(* Coast stop, Quick stop, Ramp stop *)
	IF fbProfidriveGSM.eState = E_ProfidriveGSM_State.S1_SwitchingOnInhibited THEN
		fbMoveVelocity.fTargetVelocity	:= 0;
		fbMoveVelocity.fAccMax 			:= fDecelerationCoastStop;
		fbMoveVelocity.fDecMax 			:= fDecelerationCoastStop;
	ELSIF fbProfidriveGSM.eState = E_ProfidriveGSM_State.S52_QuickStop THEN
		fbMoveVelocity.fTargetVelocity	:= 0;
		fbMoveVelocity.fAccMax 			:= fDecelerationQuickStop;
		fbMoveVelocity.fDecMax 			:= fDecelerationQuickStop;
	ELSIF fbProfidriveGSM.eState = E_ProfidriveGSM_State.S51_RampStop THEN
		fbMoveVelocity.fTargetVelocity	:= 0;
		fbMoveVelocity.fAccMax 			:= fDeceleration;
		fbMoveVelocity.fDecMax 			:= fDeceleration;
	END_IF

(* Call MoveVelocity *)
	fbMoveVelocity();
	
(* Status word *)
	stStatus.bReadyForSwitchingOn			:= fbProfidriveGSM.stStatus.b0_ReadyToSwitchOn;	
	stStatus.bReadyForOperation				:= fbProfidriveGSM.stStatus.b1_ReadyForOperation;
	stStatus.bOperationEnabled				:= stControl.bEnableOperation;
	stStatus.bFaultPresent					:= bFaultPresent;
	stStatus.bNoCoastDownActive				:= fbProfidriveGSM.eState <> E_ProfidriveGSM_State.S1_SwitchingOnInhibited;
	stStatus.bNoQuickStopActive				:= fbProfidriveGSM.eState <> E_ProfidriveGSM_State.S52_QuickStop;
	stStatus.bSwitchingOnInhibited			:= fbProfidriveGSM.stStatus.b6_SwitchingOnInhibited;
	stStatus.bAlarmPresent					:= bAlarmPresent;
	stStatus.bDeviationWithinTolerance		:= TRUE;
	stStatus.bControlRequested				:= stConfig.bControlRequested;	
	stStatus.bFrequencyLimitOk				:= TRUE;	
	stStatus.bBusy							:= ABS(fbMoveVelocity.fVelocity) > 0;
	stStatus.bInverterError					:= bInverterError;	
	stStatus.bVoltageError					:= bVoltageError;
	stStatus.bMomentError					:= bMomentError;
	stStatus.bTimerError					:= bTimerError;

(* Reset quickstop from extern *)
	IF stControl.bAcknowledgeFaults THEN
		bQuickStopExternal := FALSE;
	END_IF

(* Calculate NIST *)
	IF stConfig.fP2000 = 0 THEN
		stStatus.nIst	:= 0;
	ELSE
		stStatus.nIst	:=	REAL_TO_INT((ABS(fbMoveVelocity.fVelocity) * 16#4000) / stConfig.fP2000);
	END_IF

(* Output of actual value *)	
	IF stConfig.bOutputVelocity THEN
		ControlData := fbMoveVelocity.fVelocity;
	ELSE
		ControlData := ControlData + fbMoveVelocity.fVelocity *  GVL_Core.fbSystem.fDeltaTime * GVL_Core.fbSystem.fTimeScaling;
	END_IF
	
	fValue := ControlData;
END_METHOD

METHOD INTERNAL EvaluateParameters
VAR_INPUT
END_VAR
IF stConfig.fP1120 > 0 THEN
	fAcceleration := stConfig.fP2000/stConfig.fP1120;
ELSE
	fAcceleration := 1000;
END_IF

IF stConfig.fP1121 > 0 THEN
	fDeceleration := stConfig.fP2000/stConfig.fP1121;
ELSE
	fDeceleration := 1000;
END_IF

IF stConfig.fP1135 > 0 THEN
	fDecelerationQuickStop := stConfig.fP2000/stConfig.fP1135;
ELSE
	fDecelerationQuickStop := 1000;
END_IF

IF stConfig.fRampDownTimeCoastStop > 0 THEN
	fDecelerationCoastStop := stConfig.fP2000/stConfig.fRampDownTimeCoastStop;
ELSE
	fDecelerationCoastStop := 1000;
END_IF
END_METHOD

METHOD PUBLIC GetAcylicParameter : BOOL
VAR_INPUT
	stParameter : POINTER TO ST_PROFIdriveParam;
END_VAR
IF stParameter^.nNumber = 35 THEN
	stParameter^.nFormat := E_PROFIdriveParamFormat.FLOAT;
	stParameter^.nElements := 1;
	memcpy(ADR(stParameter^.aValue), ADR(stConfig.nR0035), 4);
END_IF
END_METHOD

METHOD INTERNAL InitRun : BOOL
VAR_INST
	bInitRun : BOOL := TRUE;
END_VAR
IF NOT bInitRun THEN RETURN; END_IF
bInitRun := FALSE;

IF pFromBus = 0 OR pToBus = 0 THEN
	ADSLOGSTR(ADSLOG_MSGTYPE_WARN, CONCAT(sPath, ': %s'), 'Plc address not set.');
END_IF
END_METHOD

METHOD INTERNAL ReadBus
VAR_INPUT
END_VAR
IF pFromBus = 0 THEN
	RETURN;
END_IF

IF NOT stConfig.bSwapProcessData THEN
	(* Control word *)
		stControl.bOFF1							:= pFromBus[0].0;
		stControl.bOFF2							:= pFromBus[0].1;
		stControl.bOFF3							:= pFromBus[0].2;
		stControl.bEnableOperation			    	:= pFromBus[0].3;
		stControl.bOperatingCondition				:= pFromBus[0].4;
		stControl.bContinueRampFunctionGenerator	:= pFromBus[0].5;
		stControl.bEnableSetpoint  				:= pFromBus[0].6;
		stControl.bAcknowledgeFaults				:= pFromBus[0].7;
		stControl.bJog1							:= pFromBus[1].0;
		stControl.bJog2							:= pFromBus[1].1;
		stControl.bDataValid						:= pFromBus[1].2;
		stControl.bFreqCorrDown					:= pFromBus[1].3;
		stControl.bFreqCorrUp						:= pFromBus[1].4;
		stControl.bParameterSelectionLSB			:= pFromBus[1].5;
		stControl.bParameterSelectionMSB			:= pFromBus[1].6;
		stControl.bReversing						:= pFromBus[1].7;
		
	(* Setpoint speed *)
		stControl.nSoll							:= UINT_TO_INT(pFromBus[2] + pFromBus[3] * 16#100);
ELSE
	(* Control word *)
		stControl.bOFF1							:= pFromBus[1].0;
		stControl.bOFF2							:= pFromBus[1].1;
		stControl.bOFF3							:= pFromBus[1].2;
		stControl.bEnableOperation				    := pFromBus[1].3;
		stControl.bOperatingCondition				:= pFromBus[1].4;
		stControl.bContinueRampFunctionGenerator	:= pFromBus[1].5;
		stControl.bEnableSetpoint  				:= pFromBus[1].6;
		stControl.bAcknowledgeFaults				:= pFromBus[1].7;
		stControl.bJog1							:= pFromBus[0].0;
		stControl.bJog2							:= pFromBus[0].1;
		stControl.bDataValid						:= pFromBus[0].2;
		stControl.bFreqCorrDown					:= pFromBus[0].3;
		stControl.bFreqCorrUp						:= pFromBus[0].4;
		stControl.bParameterSelectionLSB			:= pFromBus[0].5;
		stControl.bParameterSelectionMSB			:= pFromBus[0].6;
		stControl.bReversing						:= pFromBus[0].7;
		
	(* Setpoint speed *)
		stControl.nSoll							:= UINT_TO_INT(pFromBus[3] + pFromBus[2] * 16#100);
END_IF
END_METHOD

METHOD PUBLIC SetAcylicParameter : BOOL
VAR_INPUT
	pParameter : POINTER TO ST_PROFIdriveParam;
END_VAR
END_METHOD

METHOD PUBLIC TrigSafetyStop
bQuickStopExternal := TRUE;
END_METHOD

METHOD INTERNAL WriteBus
IF pToBus = 0 THEN
	RETURN;
END_IF

IF NOT stConfig.bSwapProcessData THEN
	(* Status word *)
		pToBus[0].0 := stStatus.bReadyForSwitchingOn			;	
		pToBus[0].1 := stStatus.bReadyForOperation				;
		pToBus[0].2 := stStatus.bOperationEnabled				;
		pToBus[0].3 := stStatus.bFaultPresent					;
		pToBus[0].4 := stStatus.bNoCoastDownActive				;
		pToBus[0].5 := stStatus.bNoQuickStopActive				;
		pToBus[0].6 := stStatus.bSwitchingOnInhibited			;
		pToBus[0].7 := stStatus.bAlarmPresent					;
		pToBus[1].0 := stStatus.bDeviationWithinTolerance		;
		pToBus[1].1 := stStatus.bControlRequested				;
		pToBus[1].2 := stStatus.bFrequencyLimitOk				;
		pToBus[1].3 := stStatus.bBusy							;
		pToBus[1].4 := stStatus.bInverterError 					;
		pToBus[1].5 := stStatus.bVoltageError					;	
		pToBus[1].6 := stStatus.bMomentError					;
		pToBus[1].7 := stStatus.bTimerError						;
	
	(* Actual speed *)
		memcpy(ADR(pToBus[3]), ADR(stStatus.nIst) + 1, 1);
		memcpy(ADR(pToBus[2]), ADR(stStatus.nIst), 1);
ELSE
	(* Status word *)
		pToBus[1].0 := stStatus.bReadyForSwitchingOn			;	
		pToBus[1].1 := stStatus.bReadyForOperation				;
		pToBus[1].2 := stStatus.bOperationEnabled				;
		pToBus[1].3 := stStatus.bFaultPresent					;
		pToBus[1].4 := stStatus.bNoCoastDownActive				;
		pToBus[1].5 := stStatus.bNoQuickStopActive				;
		pToBus[1].6 := stStatus.bSwitchingOnInhibited			;
		pToBus[1].7 := stStatus.bAlarmPresent					;
		pToBus[0].0 := stStatus.bDeviationWithinTolerance		;
		pToBus[0].1 := stStatus.bControlRequested				;
		pToBus[0].2 := stStatus.bFrequencyLimitOk				;
		pToBus[0].3 := stStatus.bBusy							;
		pToBus[0].4 := stStatus.bInverterError 					;
		pToBus[0].5 := stStatus.bVoltageError					;	
		pToBus[0].6 := stStatus.bMomentError					;
		pToBus[0].7 := stStatus.bTimerError						;
	
	(* Actual speed *)
		memcpy(ADR(pToBus[2]), ADR(stStatus.nIst) + 1, 1);
		memcpy(ADR(pToBus[3]), ADR(stStatus.nIst), 1);
END_IF
END_METHOD

END_FUNCTION_BLOCK

// ---- _backlog/ProfidriveCu/FB_ProfidriveCu.TcPOU
FUNCTION_BLOCK FB_ProfidriveCu EXTENDS FB_Base
VAR_INPUT
	stConfig 			: ST_ProfidriveCuConfig;	
	bSafetyOk			: BOOL;
END_VAR
VAR
	fbParamInterpreter	: FB_PROFIdriveParamInterpreter;
	stParamSet			: ST_PROFIdriveParamSet;
	stRecordData		: ST_AdsMessage;
	iRecordData			: I_RecordData;	
	aSinamics			: ARRAY[1..32] OF I_Sinamics; 	
	nParamState			: USINT := 0; //0=INIT 1=WRREC 2=WRRES 3=RDREC 4=RDRES
END_VAR

SUPER^();
InitRun();
Safety();
ParamStatemachine();

METHOD INTERNAL GetParam : BOOL
VAR_INPUT
	nAxisNumber : BYTE;
END_VAR

VAR	
	i : INT;	
END_VAR
GetParam := FALSE;

IF NOT IsAxisNoValid(nAxisNumber) THEN
	RETURN;
END_IF

IF fbParamInterpreter.nParameters > 0 THEN
	FOR i := 0 TO fbParamInterpreter.nParameters - 1 BY 1 DO
		aSinamics[nAxisNumber].GetAcylicParameter(ADR(stParamSet[i]));
	END_FOR
END_IF

GetParam := TRUE;
END_METHOD

METHOD INTERNAL InitRun : BOOL
VAR_INST
	bInitRun : BOOL := TRUE;
END_VAR
IF NOT bInitRun THEN RETURN; END_IF
bInitRun := FALSE;

fbParamInterpreter.pParamSet := ADR(stParamSet);

iRecordData := OC_Core.GVL_Core.fbSystem.fbRecordData;

IF iRecordData <> 0 THEN
	nParamState := 1; //WRREC	
	iRecordData.Subscribe(ADR(stConfig.stRecordIdent), stRecordData);
END_IF
END_METHOD

METHOD INTERNAL IsAxisNoValid : BOOL
VAR_INPUT
	nAxisNo	: BYTE;
END_VAR
IsAxisNoValid := nAxisNo <= 32 AND nAxisNo >= 1;
END_METHOD

METHOD INTERNAL ParamStateMachine
IF iRecordData = 0 THEN
	RETURN;
END_IF

CASE nParamState OF

1: //WRREC	
	IF iRecordData.GetWriteIndication(stRecordData) THEN
		
		(* Reset the ParamInterpreter *)
		fbParamInterpreter.Reset();
				
		(* Get/set parameters only if Axis is available *)
		IF IsAxisNoValid(stRecordData.aData[2]) THEN
			
			fbParamInterpreter(pRawData := ADR(stRecordData.aData));
			
			(* Is read command -> get parameters *)
			IF fbParamInterpreter.nCommand = 1 THEN
				GetParam(fbParamInterpreter.nAxis);
			END_IF
			
			(* Is write command -> set parameters *)
			IF fbParamInterpreter.nCommand = 2 THEN
				SetParam(fbParamInterpreter.nAxis);
			END_IF
		END_IF
		
		(* Next step is WRRES *)
		nParamState := 2;
	
	END_IF
	
2: //WRRES
	(* Send write response *)
	IF iRecordData.SendWriteResponse(stRecordData) = S_OK THEN
		(* Next step is RDREC *)
		nParamState := 3;		
	END_IF

3: //RDREC
	IF iRecordData.GetReadIndication(stRecordData) THEN		
			
		(* Make user data for response *)
		IF fbParamInterpreter.nCommand = 1 THEN
			fbParamInterpreter.MakeResponse(ADR(stRecordData.aData));
		END_IF		
		
		(* Next step is RDRES *)
		nParamState := 4;	
	END_IF
	
4: //RDRES
	(* Send read response *)
	IF iRecordData.SendReadResponse(stRecordData) = S_OK THEN
		(* Next step is WRREC *)
		nParamState := 1;		
	END_IF
	
END_CASE
END_METHOD

METHOD INTERNAL Safety : BOOL
VAR
	i : BYTE;
END_VAR
FOR i:=1 TO 32 DO
	IF aSinamics[i] <> 0 THEN
		IF NOT bSafetyOk THEN 
			aSinamics[i].TrigSafetyStop();
		END_IF
	END_IF
END_FOR
END_METHOD

METHOD INTERNAL SetParam : BOOL
VAR_INPUT
	nAxisNumber : BYTE;
END_VAR

VAR	
	i : INT;
END_VAR
SetParam := FALSE;

IF NOT IsAxisNoValid(nAxisNumber) THEN
	RETURN;
END_IF

IF fbParamInterpreter.nParameters > 0 THEN
	FOR i := 0 TO fbParamInterpreter.nParameters - 1 BY 1 DO
		aSinamics[nAxisNumber].SetAcylicParameter(ADR(stParamSet[i]));
	END_FOR
END_IF

SetParam := TRUE;
END_METHOD

METHOD PUBLIC Subscribe
VAR_INPUT
	iSinamics : I_Sinamics;
	nNumber : BYTE;
END_VAR
IF nNumber > 0 AND nNumber < 33 THEN
	aSinamics[nNumber] := iSinamics;
END_IF
END_METHOD

END_FUNCTION_BLOCK

// ---- _backlog/SEW_Movisafe_CSBx1a/FB_SEW_Movisafe_CSBx1a.TcPOU
(*
FB_SEW_Movisafe_CSBx1a simulates the funcitionaly of a SEW‑EURODRIVE MOVISAFE® module.

Disclaimer: This simulation is an independent project and is not affiliated with, endorsed by, or approved by SEW‑EURODRIVE. All rights to the SEW‑EURODRIVE brand name and trademarks remain the property of the manufacturer.
Furthermore, no guarantee is given for the completeness of the functional scope or the error-free operation of the simulation. Users should be aware that deviations from the actual product may occur.
*)

{attribute 'reflection'}
FUNCTION_BLOCK FB_SEW_Movisafe_CSBx1a EXTENDS FB_DeviceByte IMPLEMENTS I_SEW_Movisafe
VAR_INPUT	
	pControl 			: PVOID; //Pocess data from fieldbus. Size must be >= stControl.
	pStatus 			: PVOID; //Pocess data to fieldbus. Size must be >= stStatus.
	stControl 			: ST_SEW_Movisafe_CSBx1a_Control; //Control structure. Is read from the fieldbus.
	stConfig 			: ST_SEW_Movisafe_CSBx1a_Config; //Config structure. Contains parameters of the device.	

	bF_DI0				: BOOL; //State digital input 1
	bF_DI1				: BOOL; //State digital input 2
	bF_DI2				: BOOL; //State digital input 3
	bF_DI3				: BOOL; //State digital input 4
END_VAR

VAR_OUTPUT	
	stStatus			: ST_SEW_Movisafe_CSBx1a_Status;
END_VAR

VAR
    {attribute 'instance-path'} 
    {attribute 'noinit'} 
    _sPath 				: STRING; 
END_VAR

SUPER^();
InitRun();

GetControlData();
Cycle();
SetStatusData();

PROPERTY bSTO : BOOL
GET
bSTO := stStatus.b0_0_StoActive;
END_GET
END_PROPERTY

METHOD INTERNAL Cycle : BOOL
VAR_INPUT
END_VAR
stStatus.b0_0_StoActive			:= NOT stControl.b0_0_STO;
stStatus.b0_3_InputDataValid	:= TRUE;
stStatus.b0_6_Warning			:= FALSE;
stStatus.b0_7_ErrorState		:= FALSE;
stStatus.b1_0_F_DI0				:= bF_DI0;
stStatus.b1_1_F_DI1				:= bF_DI1;
stStatus.b1_2_F_DI2				:= bF_DI2;
stStatus.b1_3_F_DI3				:= bF_DI3;
stStatus.b2_2_SSx1				:= stControl.b2_2_SSx1;
stStatus.b2_3_SSx2				:= stControl.b2_3_SSx2;
END_METHOD

METHOD INTERNAL GetControlData
VAR_INPUT
END_VAR
IF pControl <= 0 OR stConfig.bForceMode THEN RETURN; END_IF

F_MEMCPY(ADR(stControl), pControl, 3, stConfig.bSwapProcessData);
END_METHOD

METHOD INTERNAL InitRun
VAR_INST
	bInitRun : BOOL := TRUE;
END_VAR
IF NOT bInitRun THEN RETURN; END_IF
bInitRun := FALSE;

IF pControl = 0 OR pStatus = 0 THEN
	ADSLOGSTR(ADSLOG_MSGTYPE_WARN, CONCAT(_sPath, ': %s'), 'Plc address not set.');
END_IF
END_METHOD

METHOD INTERNAL SetStatusData
VAR_INPUT
END_VAR
IF pStatus <= 0 THEN RETURN; END_IF

F_MEMCPY(pStatus, ADR(stStatus), 4, stConfig.bSwapProcessData);
END_METHOD

END_FUNCTION_BLOCK
